FUNCTION SPLIT_DWORD_INTO_WORDS (* this Function extracts the 2 WORD from a dword *)
  (* Standard: 61499-1; Description: Copyright (c) 2024 HR Agrartechnik GmbH This program and the accompanying materials are made available under the terms of the Eclipse Public License 2.0 which is available at https://www.eclipse.org/legal/epl-2.0/ SPDX-License-Identifier: EPL-2.0 *)
  (* Version 3.0, 2025-04-14, Patrick Aigner, changed package *)
  (* Version 1.1, 2024-07-24, Moritz Ortmeier, HR Agrartechnik, rename Function and change Output Variables *)
  (* Version 1.0, 2024-02-22, Franz Höpfinger, HR Agrartechnik, initial Implementation *)
  PACKAGE eclipse4diac::utils::splitting;
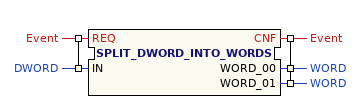
  EVENT_INPUT
    REQ WITH IN; (* Normal Execution Request *)
  END_EVENT
  EVENT_OUTPUT
    CNF WITH WORD_00, WORD_01; (* Execution Confirmation *)
  END_EVENT
  VAR_INPUT
    IN : DWORD;
  END_VAR
  VAR_OUTPUT
    WORD_00 : WORD;
    WORD_01 : WORD;
  END_VAR
  BODY IN ST:
(* this Function extracts the 2 WORD from a dword *)
FUNCTION SPLIT_DWORD_INTO_WORDS

VAR_INPUT
	IN : DWORD;
END_VAR

VAR_OUTPUT
	WORD_00 : WORD;
	WORD_01 : WORD;
END_VAR

WORD_00 := IN.%W0;
WORD_01 := IN.%W1;

END_FUNCTION
  END_BODY
END_FUNCTION
